(* IEC 61131-3 sources: s22-soft-shell/ST_resources/ST error programs, 3 files *)

(* ---- 01_bool_invalid.st ---- *)
PROGRAM 01_invalid_bool // bool should accept 0 and 1 but not any other ints
    VAR
	a : bool;
        b : bool;
        c : bool;
    END_VAR
	a := 1; //true
        a := 0; //false
        a := 5; //error!
END_PROGRAM

(* ---- 01_undeclared.st ---- *)
PROGRAM 01_undeclared  // a is being assign a value without being first declared in VARS
	a := 1;
END_PROGRAM

(* ---- 01_unknown_type.st ---- *)
PROGRAM 01_unknown_type // should error at unknown type
    VAR
	a : Foo;
    END_VAR
	a := 3.1415;
END_PROGRAM
